# EPICS substitutions: modules/event/evrSupport/Db/ioc/IOC-IN20-BP02pattern.substitutions
#
# Pattern records
file evrPatternAll.db {
#	    Device        ,  SLC Pattern Check LNK    , EVR/Trigger
#	                                                  Links
  pattern { DEVICE        ,        LINK4              , LINK5 , LINK6 , TREF    , TS1ST, TS2ND }
	  { IOC:IN20:BP02 ,"IOC:IN20:BP02:FANOUTSLC"  ,  ""   ,  ""   , 1.03E06 ,   1  ,   4   }
}
file evrEventAll.db {
  pattern { DEVICE        }
	  { IOC:IN20:BP02 }
}
